Fanuc KAREL source: NC0014.KL

-- PROVISIONAL review KL for V770-1; original PC SHA256 12b44b508866083c1ca452950fb133e3de0855c7c51a97f746095841f0ca2df2
-- Incomplete behavior may be omitted. Consult companion uncertainty JSON. Do not deploy.
PROGRAM NC0014
%NOLOCKGROUP
-- UNRESOLVED_LOCAL_POOL 1 cells at code offset 3; source declarations unknown
-- DIRECT_LOCAL_WORD_ACCESS alone does not prove INTEGER, REAL, or BOOLEAN
BEGIN
  -- UNRESOLVED_PC offsets 0-8; opcodes 2B,2C,7B
  -- UNRESOLVED_PC offsets 13-20; opcodes 9D,23
  -- UNRESOLVED_PC offsets 25-38; opcodes 21,9D,57,79
  -- UNRESOLVED_PC offsets 43-61; opcodes 21,2E,52,23
  -- UNRESOLVED_PC offsets 66-71; opcodes 7A
  -- UNRESOLVED_PC offsets 76-89; opcodes 21,9D,57,79
  -- UNRESOLVED_PC offsets 94-112; opcodes 21,2E,52,23
  -- UNRESOLVED_PC offsets 117-122; opcodes 7A
  -- UNRESOLVED_PC offsets 127-140; opcodes 21,9D,57,79
  -- UNRESOLVED_PC offsets 145-163; opcodes 21,2E,52,23
  -- UNRESOLVED_PC offsets 168-173; opcodes 7A
  -- UNRESOLVED_PC offsets 178-192; opcodes 21,9D,52,23
  -- UNRESOLVED_PC offsets 212-216; opcodes 7F
  -- UNRESOLVED_PC offsets 221-225; opcodes 27,AA
  -- UNRESOLVED_PC offsets 230-234; opcodes 7F
END NC0014
